TYPE DataStruct :
STRUCT
	bTest	: BOOL;
	nTest	: DINT;
	fTest	: LREAL;
	sTest	: STRING;
END_STRUCT
END_TYPE

(* stored: Version 1.1.0.1, ProductVersion 3.1.4026.18
   DUT DataStruct: Id {17c1d08d-d180-441c-8ec7-45defbe7d48d} *)
